{attribute 'qualified_only'}
VAR_GLOBAL
	testNonPers : INT;
END_VAR

(* stored: Version 1.1.0.1, ProductVersion 3.1.4022.12
   GVL GVL_Non_Pers: Id {4be7c746-b034-4353-8552-cb4c3cfcd6e5} *)
